// TIA Portal V17 export
// export: Created 2024-09-02T12:50:29.9857131Z, ExportSetting WithDefaults, DisplayName Totally Integrated Automation Portal, DisplayVersion V17, DisplayName TIA Portal Openness, DisplayVersion V17, DisplayName TIA Portal Version Control Interface, DisplayVersion V17, DisplayName STEP 7 Professional, DisplayVersion V17, DisplayName STEP 7 Safety, DisplayVersion V17, DisplayName WinCC Professional, DisplayVersion V17
TYPE "a_EKS"
// stored: IsFailsafeCompliant false
   STRUCT
      o_Datentraeger_Reserve_0 : Bool;
      o_Datentraeger_Reserve_1 : Bool;
      o_Datentraeger_Reserve_2 : Bool;
      o_Datentraeger_Reserve_3 : Bool;
      o_Datentraeger_Reserve_4 : Bool;
      o_Datentraeger_Reserve_5 : Bool;
      o_Datentraeger_Lesen : Bool;   // Lesekommando für Datenträger / Read command for data carrier
      o_Datentraeger_Schreiben : Bool;   // Schreibkommando für Datenträger / Write command for data carrier
      Start_Adresse : Byte;   // Start Adresse auf dem Datenträger / Start address on the data carrier
      Anzahl_Bytes : Byte;   // Anzahl der zu lesenden/schreibenden Bytes / Number of bytes to read/write
      Reserve_Byte3 : Byte;
      Sende_Daten : Array[0..11] of Char;   // zu sendende Daten fürs EKS / Data to be sent for EKS
      Reserve : Array[17..128] of Byte;   // Reserve EA / Reserve EA
   END_STRUCT;
END_TYPE
